PROGRAM HOME_MOVE
VAR
	DATA1: LREAL;
	DATAPLS : R_TRIG;
	Manual_TRIG : R_TRIG;
	AUTO_TRIG : R_TRIG;
END_VAR
//원점 순서
//1.가이드 잡고
//2.가이드 벌리고
//3. Z축 잡고 
//4. Z축 올리고
//5.Y축 잡고
//6.Y축 WAIT 포지션
//7. X 축 잡고
//8. 모두 원점 잡으면 올 WAIT 포지션

Manual_TRIG(CLK := GVL_System.Manual_Mode);
AUTO_TRIG(CLK := GVL_System.AUTO_Mode);
IF AUTO_TRIG.Q THEN
	GVL_System.All_Axis_Wait_Pos_Moving :=TRUE;
	GVL_Axis04.M_Cleaning_Move := FALSE;
END_IF
IF GVL_System.ALL_Wait_Position THEN
	GVL_System.All_Axis_Wait_Pos_Moving :=FALSE;
END_IF
IF Manual_TRIG.Q THEN
	GVL_Axis04.M_Cleaning_Move := TRUE;
	
END_IF

IF GVL_Axis04.Cleaning_Move_Position THEN
	GVL_Axis04.M_Cleaning_Move := FALSE;
END_IF

IF	(GVL_AxIS02.Wait_Position = TRUE) AND	(GVL_AxIS03.Wait_Position = TRUE) AND	(GVL_AxIS04.Wait_Position = TRUE) AND (GVL_AxIS05.Wait_Position = TRUE) THEN
	
		GVL_System.ALL_Wait_Position := TRUE;
	
ELSE
		GVL_System.ALL_Wait_Position := FALSE;
	
END_IF


IF GVL_SYSTEM.ALL_Home_Move_PB = TRUE AND GVL_System.Manual_Mode = TRUE  AND (GVL_System.ALL_Motor_Homed = FALSE) THEN
	
	GVL_SYSTEM.ALL_Home_Move_Start := TRUE;		// 원점 시작
	
	GVL_Axis01.Wait_Position_Data := 38;
	
END_IF

IF	(GVL_System.ALL_Home_Move_Start = TRUE) THEN
	
	GVL_System.Axis04_Home_Move := TRUE;	// Z축 원점 시작
	
	IF (GVL_Axis04.Home_OK = TRUE) THEN
		
		GVL_System.Axis02_Home_Move := TRUE;	     //Z축 원점 확인 후 X축 원점 시작  //
		
	END_IF
	IF (GVL_Axis02.Home_OK = TRUE) THEN
		
		GVL_System.Axis01_Home_Move := TRUE;
		GVL_System.Axis03_Home_Move := TRUE;	//   X축 원점 확인 후 가이드 Y,R 축 모두 원점 시작 GVL_System.Axis04_Home_Move
		
	END_IF
	IF (GVL_Axis01.Home_OK = TRUE) THEN
		GVL_System.Axis01_Wait_Pos_Move  := TRUE ;
	END_IF
	IF (GVL_Axis03.Home_OK = TRUE) THEN
		GVL_System.Axis05_Home_Move := TRUE;
	END_IF
	
		
	
	IF	(GVL_System.ALL_Motor_Homed = TRUE) AND (GVL_Axis01.Wait_Position = TRUE)  THEN
		//모든 측 원점 확인 후 리셋 및 wait 포지션 이동
		
		GVL_SYSTEM.Axis01_Home_Move := FALSE;
		GVL_SYSTEM.Axis02_Home_Move := FALSE;
		GVL_SYSTEM.Axis03_Home_Move := FALSE;
		GVL_SYSTEM.Axis04_Home_Move := FALSE;
		GVL_SYSTEM.Axis05_Home_Move := FALSE;
		GVL_System.Axis01_Wait_Pos_Move := FALSE;
		
		GVL_SYSTEM.Axis02_Wait_Pos_Move := TRUE;
		GVL_SYSTEM.Axis03_Wait_Pos_Move := TRUE;
		GVL_SYSTEM.Axis04_Wait_Pos_Move := TRUE;
		GVL_SYSTEM.Axis05_Wait_Pos_Move := TRUE;
	
	END_IF
	IF	(GVL_System.ALL_Wait_Position = TRUE) THEN
		
		GVL_SYSTEM.ALL_Home_Move_Start 	:= FALSE;
		GVL_SYSTEM.Axis02_Wait_Pos_Move := FALSE;
		GVL_SYSTEM.Axis03_Wait_Pos_Move := FALSE;
		GVL_SYSTEM.Axis04_Wait_Pos_Move := FALSE;
		GVL_SYSTEM.Axis05_Wait_Pos_Move := FALSE;
	END_IF

END_IF

END_PROGRAM

(* stored: Version 1.1.0.1, ProductVersion 3.1.4024.15
   POU HOME_MOVE: Id {0b7a5dc2-9791-47fe-9b1f-c3a35a108549}, SpecialFunc None *)
